// LS Electric XG5000 project: SeletoraCodLadder
// PLC NewPLC
// module base 0 slot 1: FEnet:XBL-EMTA

PROGRAM Main (task: Scan Program)

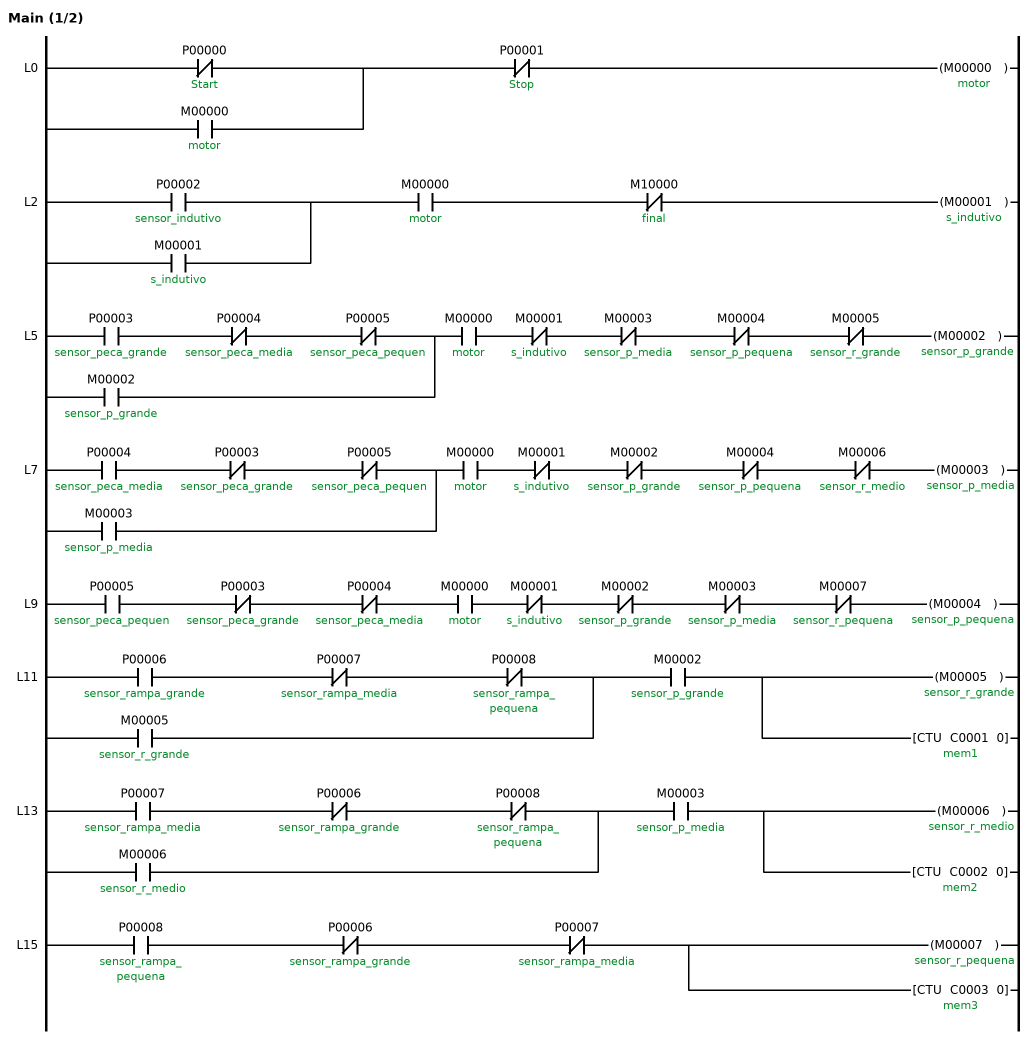
; L0
LOAD NOT  P00000	// Start
OR        M00000	// motor
AND NOT   P00001	// Stop
OUT       M00000	// motor
; L2
LOAD      P00002	// sensor_indutivo
OR        M00001	// s_indutivo
AND       M00000	// motor
AND NOT   M10000	// final
OUT       M00001	// s_indutivo
; L5
LOAD      P00003	// sensor_peca_grande
AND NOT   P00004	// sensor_peca_media
AND NOT   P00005	// sensor_peca_pequen
OR        M00002	// sensor_p_grande
AND       M00000	// motor
AND NOT   M00001	// s_indutivo
AND NOT   M00003	// sensor_p_media
AND NOT   M00004	// sensor_p_pequena
AND NOT   M00005	// sensor_r_grande
OUT       M00002	// sensor_p_grande
; L7
LOAD      P00004	// sensor_peca_media
AND NOT   P00003	// sensor_peca_grande
AND NOT   P00005	// sensor_peca_pequen
OR        M00003	// sensor_p_media
AND       M00000	// motor
AND NOT   M00001	// s_indutivo
AND NOT   M00002	// sensor_p_grande
AND NOT   M00004	// sensor_p_pequena
AND NOT   M00006	// sensor_r_medio
OUT       M00003	// sensor_p_media
; L9
LOAD      P00005	// sensor_peca_pequen
AND NOT   P00003	// sensor_peca_grande
AND NOT   P00004	// sensor_peca_media
AND       M00000	// motor
AND NOT   M00001	// s_indutivo
AND NOT   M00002	// sensor_p_grande
AND NOT   M00003	// sensor_p_media
AND NOT   M00007	// sensor_r_pequena
OUT       M00004	// sensor_p_pequena
; L11
LOAD      P00006	// sensor_rampa_grande
AND NOT   P00007	// sensor_rampa_media
AND NOT   P00008	// sensor_rampa_pequena
OR        M00005	// sensor_r_grande
AND       M00002	// sensor_p_grande
OUT       M00005	// sensor_r_grande
CTU       C0001 0	// mem1
; L13
LOAD      P00007	// sensor_rampa_media
AND NOT   P00006	// sensor_rampa_grande
AND NOT   P00008	// sensor_rampa_pequena
OR        M00006	// sensor_r_medio
AND       M00003	// sensor_p_media
OUT       M00006	// sensor_r_medio
CTU       C0002 0	// mem2
; L15
LOAD      P00008	// sensor_rampa_pequena
AND NOT   P00006	// sensor_rampa_grande
AND NOT   P00007	// sensor_rampa_media
OUT       M00007	// sensor_r_pequena
CTU       C0003 0	// mem3

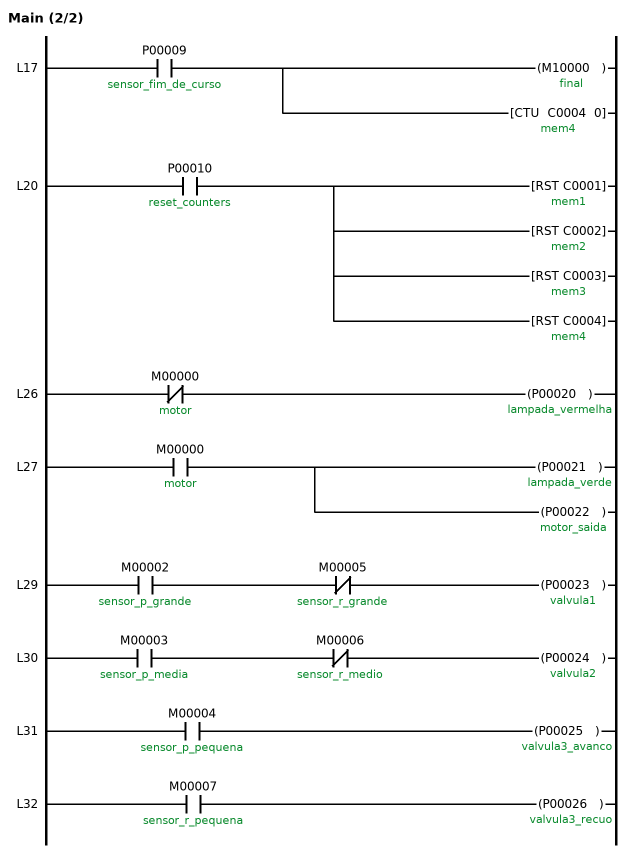
; L17
LOAD      P00009	// sensor_fim_de_curso
OUT       M10000	// final
CTU       C0004 0	// mem4
; L20
LOAD      P00010	// reset_counters
RST       C0001	// mem1
RST       C0002	// mem2
RST       C0003	// mem3
RST       C0004	// mem4
; L26
LOAD NOT  M00000	// motor
OUT       P00020	// lampada_vermelha
; L27
LOAD      M00000	// motor
OUT       P00021	// lampada_verde
OUT       P00022	// motor_saida
; L29
LOAD      M00002	// sensor_p_grande
AND NOT   M00005	// sensor_r_grande
OUT       P00023	// valvula1
; L30
LOAD      M00003	// sensor_p_media
AND NOT   M00006	// sensor_r_medio
OUT       P00024	// valvula2
; L31
LOAD      M00004	// sensor_p_pequena
OUT       P00025	// valvula3_avanco
; L32
LOAD      M00007	// sensor_r_pequena
OUT       P00026	// valvula3_recuo

VARIABLES AND COMMENTS (devices not used above)
P00011	BIT	res